// Mitsubishi GX Works2 project: 240517_A+B+B-A-C+C-카운트   PLC: Q02U

PROGRAM MAIN
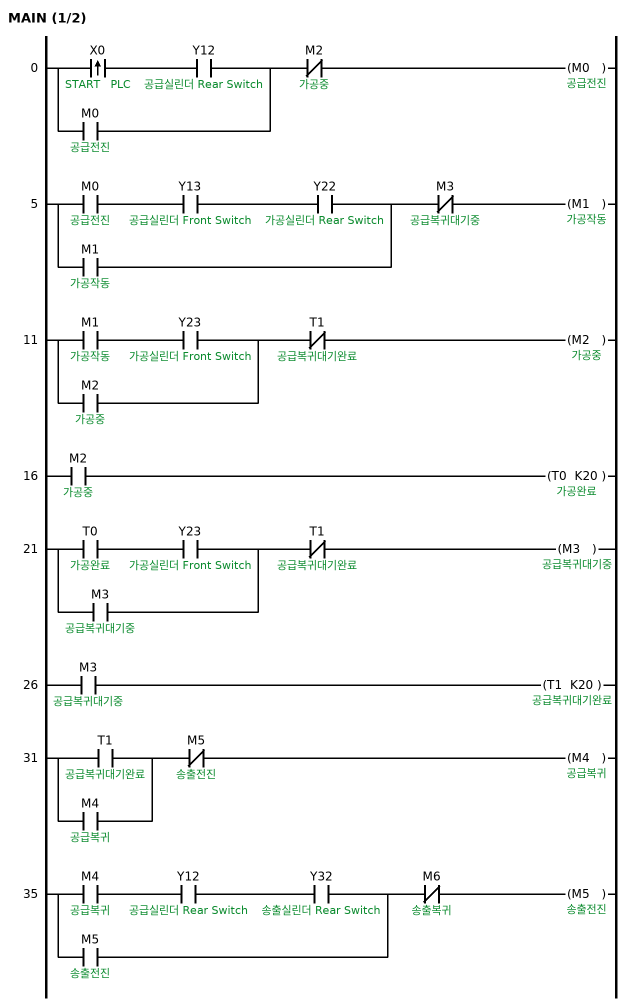
0     LDP     X0  ; START   PLC
      AND     Y12  ; 공급실린더 Rear Switch
      OR      M0  ; 공급전진
      ANI     M2  ; 가공중
      OUT     M0  ; 공급전진
5     LD      M0  ; 공급전진
      AND     Y13  ; 공급실린더 Front Switch
      AND     Y22  ; 가공실린더 Rear Switch
      OR      M1  ; 가공작동
      ANI     M3  ; 공급복귀대기중
      OUT     M1  ; 가공작동
11    LD      M1  ; 가공작동
      AND     Y23  ; 가공실린더 Front Switch
      OR      M2  ; 가공중
      ANI     T1  ; 공급복귀대기완료
      OUT     M2  ; 가공중
16    LD      M2  ; 가공중
      OUT     T0 K20  ; 가공완료
21    LD      T0  ; 가공완료
      AND     Y23  ; 가공실린더 Front Switch
      OR      M3  ; 공급복귀대기중
      ANI     T1  ; 공급복귀대기완료
      OUT     M3  ; 공급복귀대기중
26    LD      M3  ; 공급복귀대기중
      OUT     T1 K20  ; 공급복귀대기완료
31    LD      T1  ; 공급복귀대기완료
      OR      M4  ; 공급복귀
      ANI     M5  ; 송출전진
      OUT     M4  ; 공급복귀
35    LD      M4  ; 공급복귀
      AND     Y12  ; 공급실린더 Rear Switch
      AND     Y32  ; 송출실린더 Rear Switch
      OR      M5  ; 송출전진
      ANI     M6  ; 송출복귀
      OUT     M5  ; 송출전진
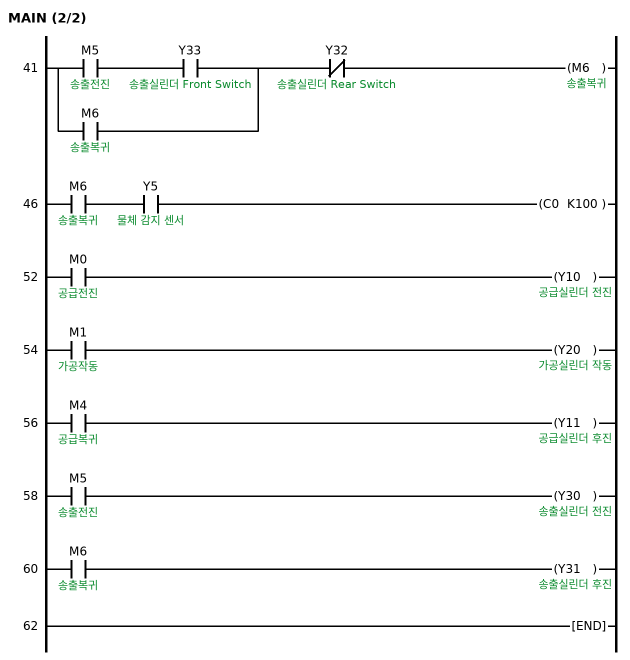
41    LD      M5  ; 송출전진
      AND     Y33  ; 송출실린더 Front Switch
      OR      M6  ; 송출복귀
      ANI     Y32  ; 송출실린더 Rear Switch
      OUT     M6  ; 송출복귀
46    LD      M6  ; 송출복귀
      AND     Y5  ; 물체 감지 센서
      OUT     C0 K100
52    LD      M0  ; 공급전진
      OUT     Y10  ; 공급실린더 전진
54    LD      M1  ; 가공작동
      OUT     Y20  ; 가공실린더 작동
56    LD      M4  ; 공급복귀
      OUT     Y11  ; 공급실린더 후진
58    LD      M5  ; 송출전진
      OUT     Y30  ; 송출실린더 전진
60    LD      M6  ; 송출복귀
      OUT     Y31  ; 송출실린더 후진
62    END
END_PROGRAM

// device comments not shown above
X1  ; STOP PLC
X10  ; 공급    Rear    Switch
X11  ; 공급    Front   Switch
Y0  ; 컨베이어
Y1  ; RED LAMP
Y2  ; YELLOW LAMP
Y3  ; GREEN LAMP
Y4  ; 공급 감지 센서
Y6  ; 금속 감지 센서
Y40  ; 배출출실린더 전진
Y41  ; 배출실린더 후진
Y42  ; 배출실린더 Rear Switch
Y43  ; 배출실린더 Front Switch
